{attribute 'qualified_only'}
{attribute 'strict'}
TYPE E_RobotTaskStates :
(
	Idle,
	TaskTypeSelection,
	TaskSelection,
	TaskAssignment,
	TaskAssignment_Wait,
	TaskExecution
);
END_TYPE

(* stored: Version 1.1.0.1, ProductVersion 3.1.4020.12
   DUT E_RobotTaskStates: Id {f658457b-6584-47e2-8259-9b1ccee486ea} *)
